TYPE ST_Rectify :   //纠偏控制
STRUCT
(********参数**************)	

	bReset            :BOOL;     // 纠偏复位  
	bEnable		:BOOL;	(*开启自动纠偏*)
	fSensorActValue			:REAL; //实际位置
	
	bReady              :BOOL;  //纠偏准备号
	bAutoRunning		:BOOL;	(*纠偏自动运行中*)
	Error		:BOOL;            //纠偏错误
    ErrID:	 STRING;     //纠偏错误代码
	
END_STRUCT
END_TYPE

(* stored: Version 1.1.0.1, ProductVersion 3.1.4024.9
   DUT ST_Rectify: Id {09ecaf26-9a3e-4d9a-b68f-e6c36b49f428} *)
